// TIA Portal V20 export
FUNCTION_BLOCK "FB_McpKeyboardSignals"   // FB420, SCL
{ S7_Optimized_Access := 'TRUE' }
// stored: AutoNumber false, MemoryReserve 100, SetENOAutomatically false
   VAR
      sK1_Powermeter : "FB_McpKeysSignals";
      sK2_GasAssist : "FB_McpKeysSignals";
      sK3_KeySaveParam : "FB_McpKeysSignals";
      sK4_GripperUndrilledPart : "FB_McpKeysSignals";
      sK5_GripperDrilledPart : "FB_McpKeysSignals";
      sK6_SITestStop : "FB_McpKeysSignals";
      sK7_FixtureClamp : "FB_McpKeysSignals";
      sK8_FixtureVacuum : "FB_McpKeysSignals";
      sK9_Aspiration : "FB_McpKeysSignals";
      sK10_LoaderAuto : "FB_McpKeysSignals";
      sK11_LoaderSemiAuto : "FB_McpKeysSignals";
      sK12_ObservationCamera : "FB_McpKeysSignals";
      sK13_MainDoor : "FB_McpKeysSignals";
      sK14_WarmUp : "FB_McpKeysSignals";
      sK15_MachineLight : "FB_McpKeysSignals";
      sStartCycle { S7_SetPoint := 'True'} : "FB_McpKeysSignals";
      sAlarmReset { S7_SetPoint := 'True'} : "FB_McpKeysSignals";
      sPowerOFF { S7_SetPoint := 'True'} : "FB_McpKeysSignals";
      sShutdownPC { S7_SetPoint := 'True'} : "FB_McpKeysSignals";
      sLightTest { S7_SetPoint := 'True'} : "FB_McpKeysSignals";
      sPowerON { S7_SetPoint := 'True'} : "FB_McpKeysSignals";
      sRemoteOpenShutter { S7_SetPoint := 'True'} : "FB_McpKeysSignals";
      sAx10_LaserArea { S7_SetPoint := 'True'} : "FB_McpKeysSignals";
      sAx11_ChannelSelection { S7_SetPoint := 'True'} : "FB_McpKeysSignals";
   END_VAR
   VAR_TEMP
      tNoLed : Bool;   // Index for loop
   END_VAR
BEGIN
   REGION Description header 
       //==================================================================================
       // POSALUX Swiss SA / (C) Copyright 2024
       //----------------------------------------------------------------------------------
       // Title: Management of inputs and outputs for MCP buttons
       // Comment/Function: 
       //
       // Author: Gowsigan SRITHARAN
       // Engineering: TIA Portal v17
       //----------------------------------------------------------------------------------
       // Change log table:
       // Version  | Date     | Expert in charge | Changes applied
       // ---------|----------|------------------|------------------------------------
       // 00.00.01 | 20241120 | GSR              | First released version
       // 00.00.02 | 20250911 | WFA              | PB - LED Management with multi-instance FB
       // ==================================================================================
   END_REGION

   REGION Customer keys (Middle panel)
       // Key1 : Powermeter
       #sK1_Powermeter(iKeyHWStatus := "MCP1_In".customerKey1,
                       oLedHWStatus =>"MCP1_Out".LEDcustomerKey1);

       // Key2 : Gas Assist
       #sK2_GasAssist(iKeyHWStatus := "MCP1_In".customerKey2,
                      oLedHWStatus => "MCP1_Out".LEDcustomerKey2);

       // Key3 : Save Param
       #sK3_KeySaveParam(iKeyHWStatus := "MCP1_In".customerKey3,
                         oLedHWStatus => "MCP1_Out".LEDcustomerKey3);

       // Key4 : Gripper Undrilled Part
       #sK4_GripperUndrilledPart(iKeyHWStatus := "MCP1_In".customerKey4,
                                 oLedHWStatus => "MCP1_Out".LEDcustomerKey4);

       // Key5 : Gripper Drilled Part
       #sK5_GripperDrilledPart(iKeyHWStatus := "MCP1_In".customerKey5,
                               oLedHWStatus => "MCP1_Out".LEDcustomerKey5);

       // Key6 : SI Test Stop
       #sK6_SITestStop(iKeyHWStatus := "MCP1_In".customerKey6,
                       oLedHWStatus => "MCP1_Out".LEDcustomerKey6);

       // Key7 : Fixture Clamp
       #sK7_FixtureClamp(iKeyHWStatus := "MCP1_In".customerKey7,
                         oLedHWStatus => "MCP1_Out".LEDcustomerKey7);

       // Key8 : Fixture Vacuum
       #sK8_FixtureVacuum(iKeyHWStatus := "MCP1_In".customerKey8,
                          oLedHWStatus => "MCP1_Out".LEDcustomerKey8);

       // Key9 : Aspiration
       #sK9_Aspiration(iKeyHWStatus := "MCP1_In".customerKey9,
                       oLedHWStatus => "MCP1_Out".LEDcustomerKey9);

       // Key10 : Loader Mode Auto
       #sK10_LoaderAuto(iKeyHWStatus := "MCP1_In".customerKey10,
                        oLedHWStatus => "MCP1_Out".LEDcustomerKey10);

       // Key11 : Loader Mode Semi Auto
       #sK11_LoaderSemiAuto(iKeyHWStatus := "MCP1_In".customerKey11,
                            oLedHWStatus => "MCP1_Out".LEDcustomerKey11);

       // Key12 : Observation Camera
       #sK12_ObservationCamera(iKeyHWStatus := "MCP1_In".customerKey12,
                               oLedHWStatus => "MCP1_Out".LEDcustomerKey12);

       // Key13 : Main Door
       #sK13_MainDoor(iKeyHWStatus := "MCP1_In".customerKey13,
                      oLedHWStatus => "MCP1_Out".LEDcustomerKey13);

       // Key14 : Warm Up
       #sK14_WarmUp(iKeyHWStatus := "MCP1_In".customerKey14,
                    oLedHWStatus => "MCP1_Out".LEDcustomerKey14);

       // Key15 : Camera Light
       #sK15_MachineLight(iKeyHWStatus := "MCP1_In".customerKey15,
                          oLedHWStatus => "MCP1_Out".LEDcustomerKey15);
   END_REGION Customer keys    

   REGION External Keys /LED
       // Start Cycle
       #sStartCycle(iKeyHWStatus := "DI_PB_StartCycle",
                    oLedHWStatus => "DQ_StartCycleGreenLED");

       // Alarm Reset
       #sAlarmReset(iKeyHWStatus := "DI_PB_ResetAlarm",
                    oLedHWStatus => "DQ_AlarmBlueLED");

       // Power OFF
       #sPowerOFF(iKeyHWStatus := "DI_PB_PowerOFF",
                  oLedHWStatus => #tNoLed);

       // Shutdown PC
       #sShutdownPC(iKeyHWStatus := "DI_PB_ShutdownPC",
                    oLedHWStatus => "DQ_ShutdownPCYellowLED");

       // Light Test
       #sLightTest(iKeyHWStatus := "DI_PB_LightTest",
                   oLedHWStatus => "DQ_LightTestWhiteLED");

       // Power ON
       #sPowerON(iKeyHWStatus := "DI_PB_PowerON",
                 oLedHWStatus => "DQ_PowerOnGreenLED");

       // Remote Open Shutter
       #sRemoteOpenShutter(iKeyHWStatus := "DI_PB_RemoteOpenShutter",
                           oLedHWStatus => "DQ_RemoteOpenShutterWhiteLED");
   END_REGION

   REGION Axis Keys (Right Panel)
       #sAx10_LaserArea(iKeyHWStatus := "MCP1_In".axis10,
                        oLedHWStatus => "MCP1_Out".LEDaxis10);

       #sAx11_ChannelSelection(iKeyHWStatus := "MCP1_In".axis11,
                               oLedHWStatus => "MCP1_Out".LEDaxis11);
   END_REGION
END_FUNCTION_BLOCK
